--- Backups/vIRB4600-40-2.55-RW11/RAPID/TASK3/SYSMOD/RRC_Control_Rx.sys ---
MODULE RRC_Control_Rx(SYSMODULE)
    !***********************************************************************************
    !
    ! ETH Zurich / Robotic Fabrication Lab
    ! HIB C 13 / Stefano-Franscini-Platz 1
    ! CH-8093 Zurich
    !
    !***********************************************************************************
    !
    ! PROJECT     :  RRC - Rapid Robot Communication
    !
    ! FUNCTION    :  Control modul for the project
    !
    ! AUTHOR      :  Philippe Fleischmann
    !
    ! EMAIL       :  rrc@arch.ethz.ch
    !
    ! HISTORY     :  2019.02.22
    !
    ! Copyright   :  ETH Zurich (CH) 2019
    !                - Philippe Fleischmann
    !                - Michael Lyrenmann
    !                - Gonzalo Casas
    !
    ! License     :  This code base is governed by an EULA (End-User License Agreement)
    !                which you have received together with the software.
    !                You are not allowed to use the software on a real robots
    !                without a signed EULA.
    !
    !                A copy of the EULA content is in the controller task (T_CTRL).
    !
    !***********************************************************************************

    !************************************************
    ! Function    :     Main for Project RRC
    ! Programmer  :     Philippe Fleischmann
    ! Date        :     2019.02.22
    !***************** ETH Zurich *******************
    !
    PROC r_RRC_Main()
        !
        ! Wait until controller has set taskliste all
        WaitTime n_RRC_TimeTaskLiAll;
        !
        ! Task synchronisation
        WaitSyncTask id_RRC_MainSta,tl_RRC_All;
        !
        ! Message for Operator
        TPWrite "RRC Main";
        !
        ! Initialize cell
        r_RRC_InitCell;
        !
        ! Work process
        WHILE b_RRC_Run=TRUE DO
            !
            ! Check and receive data from client 1
            IF b_RRC_Com{n_RRC_R1_ChaNr}=TRUE r_RRC_CheckAndRecFrmClient n_RRC_R1_ChaNr;
            !
            ! Check and receive data from client 2
            IF b_RRC_Com{n_RRC_R2_ChaNr}=TRUE r_RRC_CheckAndRecFrmClient n_RRC_R2_ChaNr;
            !
            ! Check and receive data from client 3
            IF b_RRC_Com{n_RRC_R3_ChaNr}=TRUE r_RRC_CheckAndRecFrmClient n_RRC_R3_ChaNr;
            !
            ! Check and receive data from client 4
            IF b_RRC_Com{n_RRC_R4_ChaNr}=TRUE r_RRC_CheckAndRecFrmClient n_RRC_R4_ChaNr;
            !
            ! Check cycle time stop watch activ
            IF b_RRC_EvLogMsgInUntilMsgOutTime=TRUE THEN
                !
                ! Measure cycle time
                IF b_RRC_FeedbackOut=TRUE THEN
                    !
                    ! Reset variable
                    b_RRC_FeedbackOut:=FALSE;
                    !
                    ! Stop read message input to feedback done watch
                    ClkStop clk_RRC_MsgInUntilMsgOut;
                    !
                    ! Log current read and unpack time in RobotStudio output
                    r_RRC_EvLogMsg st_RRC_EvLogMsgHeader,"Msg in until Msg out time : "+NumToStr(ClkRead(clk_RRC_MsgInUntilMsgOut\HighRes),3);
                ENDIF
            ENDIF
        ENDWHILE
        !
        ! Message for Operator
        TPWrite "RRC End";
        !
        ! Task synchronisation
        WaitSyncTask id_RRC_MainEnd,tl_RRC_All;
        !
        RETURN ;
    ERROR
        ! Placeholder for Error Code...
    ENDPROC

    !************************************************
    ! Function    :     Initialize Cell
    ! Programmer  :     Philippe Fleischmann
    ! Date        :     2019.02.22
    !***************** ETH Zurich *******************
    !
    PROC r_RRC_InitCell()
        !
        ! Task synchronisation
        WaitSyncTask id_RRC_InitSta,tl_RRC_All;
        !
        ! Task synchronisation wait for controller data
        WaitSyncTask id_RRC_InitCtrl,tl_RRC_All;
        !
        ! Initialize variables
        r_RRC_InitVar;
        !
        ! Initalize protocol log
        !* r_RRC_LogProtInit;
        !
        ! Initialize sockets
        IF b_RRC_SocketActiv=TRUE r_RRC_InitSockets;
        !
        ! Task synchronisation
        WaitSyncTask id_RRC_InitEnd,tl_RRC_All;
        RETURN ;
    ERROR
        ! Placeholder for Error Code...
    ENDPROC

    !************************************************
    ! Function    :     Initialize Variables
    ! Programmer  :     Philippe Fleischmann
    ! Date        :     2019.02.22
    !***************** ETH Zurich *******************
    !
    PROC r_RRC_InitVar()
        !
        ! Set Task on
        b_RRC_TaskReceiverOn:=TRUE;
        !
        ! Reset buffer full bits controller
        b_RRC_BufFullMa{n_RRC_R1_ChaNr}:=FALSE;
        b_RRC_BufFullMa{n_RRC_R2_ChaNr}:=FALSE;
        b_RRC_BufFullMa{n_RRC_R3_ChaNr}:=FALSE;
        b_RRC_BufFullMa{n_RRC_R4_ChaNr}:=FALSE;
        !
        ! Reset buffer full bits robot
        b_RRC_BufFullRob{n_RRC_R1_ChaNr}:=FALSE;
        b_RRC_BufFullRob{n_RRC_R2_ChaNr}:=FALSE;
        b_RRC_BufFullRob{n_RRC_R3_ChaNr}:=FALSE;
        b_RRC_BufFullRob{n_RRC_R4_ChaNr}:=FALSE;
        !
        ! Set first cycle bools
        b_RRC_FirstProtocolAfterPPMain:=TRUE;
        !
        ! Temp to measure cycle time
        b_RRC_FeedbackOut:=FALSE;
        !
        ! Reset counters controller
        n_RRC_WritePtrBufCtrl{n_RRC_R1_ChaNr}:=0;
        n_RRC_WritePtrBufCtrl{n_RRC_R2_ChaNr}:=0;
        n_RRC_WritePtrBufCtrl{n_RRC_R3_ChaNr}:=0;
        n_RRC_WritePtrBufCtrl{n_RRC_R4_ChaNr}:=0;
        !
        ! Reset counters robot
        n_RRC_WritePtrBufRob{n_RRC_R1_ChaNr}:=0;
        n_RRC_WritePtrBufRob{n_RRC_R2_ChaNr}:=0;
        n_RRC_WritePtrBufRob{n_RRC_R3_ChaNr}:=0;
        n_RRC_WritePtrBufRob{n_RRC_R4_ChaNr}:=0;
        !
        ! Clear buffer controller
        FOR i FROM 1 TO DIM(bm_RRC_RecBufferCtrl,2) DO
            !
            ! Overwrite with an empty message
            bm_RRC_RecBufferCtrl{n_RRC_R1_ChaNr,i}:=bmEmpty;
            bm_RRC_RecBufferCtrl{n_RRC_R2_ChaNr,i}:=bmEmpty;
            bm_RRC_RecBufferCtrl{n_RRC_R3_ChaNr,i}:=bmEmpty;
            bm_RRC_RecBufferCtrl{n_RRC_R4_ChaNr,i}:=bmEmpty;
            !
        ENDFOR
        !
        ! Clear buffer robots
        FOR i FROM 1 TO DIM(bm_RRC_RecBufferRob,2) DO
            !
            ! Overwrite with an empty message
            bm_RRC_RecBufferRob{n_RRC_R1_ChaNr,i}:=bmEmpty;
            bm_RRC_RecBufferRob{n_RRC_R2_ChaNr,i}:=bmEmpty;
            bm_RRC_RecBufferRob{n_RRC_R3_ChaNr,i}:=bmEmpty;
            bm_RRC_RecBufferRob{n_RRC_R4_ChaNr,i}:=bmEmpty;
            !
        ENDFOR
        !
        ! Reset expected Sequince ID
        n_RRC_SIDExpected{n_RRC_R1_ChaNr}:=0;
        n_RRC_SIDExpected{n_RRC_R2_ChaNr}:=0;
        n_RRC_SIDExpected{n_RRC_R3_ChaNr}:=0;
        n_RRC_SIDExpected{n_RRC_R4_ChaNr}:=0;
        RETURN ;
    ERROR
        ! Placeholder for Error Code...
    ENDPROC

    !************************************************
    ! Function    :     ProgError
    ! Programmer  :     Philippe Fleischmann
    ! Date        :     2019.02.22
    !***************** ETH Zurich *******************
    !
    PROC r_RRC_ProgError()
        !
        ! User Info
        TPWrite "Program Error";
        !
        ! Stop Program
        Stop;
        RETURN ;
    ERROR
        ! Placeholder for Error Code...
    ENDPROC

ENDMODULE

--- Backups/vIRB4600-40-2.55-RW11/RAPID/TASK3/SYSMOD/RRC_DataTask_Rx.sys ---
MODULE RRC_DataTask_Rx(SYSMODULE)
    !***********************************************************************************
    !
    ! ETH Zurich / Robotic Fabrication Lab
    ! HIB C 13 / Stefano-Franscini-Platz 1
    ! CH-8093 Zurich
    !
    !***********************************************************************************
    !
    ! PROJECT     :  RRC - Rapid Robot Communication
    !
    ! FUNCTION    :  Includ all Task specific Data's
    !
    ! AUTHOR      :  Philippe Fleischmann
    !
    ! EMAIL       :  rrc@arch.ethz.ch
    !
    ! HISTORY     :  2019.02.22
    !
    ! Copyright   :  ETH Zurich (CH) 2019
    !                - Philippe Fleischmann
    !                - Michael Lyrenmann
    !                - Gonzalo Casas
    !
    ! License     :  This code base is governed by an EULA (End-User License Agreement)
    !                which you have received together with the software.
    !                You are not allowed to use the software on a real robots
    !                without a signed EULA.
    !
    !                A copy of the EULA content is in the controller task (T_CTRL).
    !
    !***********************************************************************************

    !************************************************
    ! Declaration :     bool
    !************************************************
    !
    CONST bool b_RRC_Run:=TRUE;
    !
    TASK PERS bool b_RRC_SocketActiv:=TRUE;
    TASK PERS bool b_RRC_PrintPrio1:=FALSE;
    TASK PERS bool b_RRC_PrintPrio2:=FALSE;
    !
    TASK PERS bool b_RRC_BufFullMa{n_RRC_NumOfCha}:=[FALSE,FALSE,FALSE,FALSE];
    TASK PERS bool b_RRC_BufFullRob{n_RRC_NumOfCha}:=[FALSE,FALSE,FALSE,FALSE];
    TASK PERS bool b_RRC_LogHelper{n_RRC_NumOfCha}:=[FALSE,FALSE,FALSE,FALSE];
    !
    TASK PERS bool b_RRC_FirstProtocolAfterPPMain:=FALSE;

    !************************************************
    ! Declaration :     num
    !************************************************
    !
    CONST num n_RRC_NumOfCha:=4;
    CONST num n_RRC_RecMinData:=49;
    CONST num n_RRC_NoOfByMsgLen:=4;
    CONST num n_RRC_TimeOutRecRobSocRec:=10;
    !
    TASK PERS num n_RRC_WritePtrBufCtrl{n_RRC_NumOfCha}:=[0,0,0,0];
    TASK PERS num n_RRC_WritePtrBufRob{n_RRC_NumOfCha}:=[7,0,0,0];
    TASK PERS num n_RRC_SIDExpected{n_RRC_NumOfCha}:=[1,0,0,0];
    TASK PERS num n_RRC_SIDIs{n_RRC_NumOfCha}:=[70001,0,0,0];
    !
    VAR num n_RRC_MsgLenRob{n_RRC_NumOfCha};
    VAR num n_RRC_NoOfRecBytesRob{n_RRC_NumOfCha};

    !************************************************
    ! Declaration :     string
    !************************************************
    !
    TASK PERS string st_RRC_EvLogMsgHeader:="RRC -- Receiver";
    TASK PERS string st_RRC_SIDRestart:="S-ID User code restarted";
    !
    TASK PERS string st_RRC_UIAnswer:="Stop";
    TASK PERS string st_RRC_ActMsg1:="Expected protocol version: 1.0";
    TASK PERS string st_RRC_ActMsg2:="Received protocol version: 2.0";
    TASK PERS string st_RRC_ActMsg3:="Expected: 2";
    TASK PERS string st_RRC_ActMsg4:="Received: 70001";
    TASK PERS string st_RRC_ActMsg5:="";
    TASK PERS string st_RRC_ActBtn1:="Stop";
    TASK PERS string st_RRC_ActBtn2:="100 mm/s";
    TASK PERS string st_RRC_ActBtn3:="Set my Speed";
    TASK PERS string st_RRC_ActBtn4:="";
    TASK PERS string st_RRC_ActBtn5:="";
    TASK PERS string st_RRC_Header:="Protocol mismatch";
    !
    VAR string st_RRC_IP_ClientRec{n_RRC_NumOfCha}:=["","","",""];

    !************************************************
    ! Declaration :     clock
    !************************************************
    !
    VAR clock clk_RRC_ReadAndUnpack;
    VAR clock clk_RRC_MsgInUntilMsgOut;

    !************************************************
    ! Declaration :     RRC_Protokol
    !************************************************
    !
    CONST RRC_Protocol pro_RRC_Empty:=[[0,0,0,0],[0,0,0,"",0,0,"",0,0,0,"",0,"",0,"",0,"",0,"",0,"",0,"",0,"",0,0,0,0,0,0,0,0,0,0,0,0,0,0,0,0,0,0,0,0,0,0,0,0,0,0,0,0,0,0,0,0,0,0,0,0,0]];
    !
    VAR RRC_Protocol pro_RRC_ActMsgRob:=[[0,0,0,0],[0,0,0,"",0,0,"",0,0,0,"",0,"",0,"",0,"",0,"",0,"",0,"",0,"",0,0,0,0,0,0,0,0,0,0,0,0,0,0,0,0,0,0,0,0,0,0,0,0,0,0,0,0,0,0,0,0,0,0,0,0,0]];
    !
    TASK PERS RRC_Protocol pro_RRC_ActMsgTemp:=[[0,0,0,0],[0,0,0,"",0,0,"",0,0,0,"",0,"",0,"",0,"",0,"",0,"",0,"",0,"",0,0,0,0,0,0,0,0,0,0,0,0,0,0,0,0,0,0,0,0,0,0,0,0,0,0,0,0,0,0,0,0,0,0,0,0,0]];
    !
    TASK PERS RRC_Protocol pro_RRC_ActMsgRec{n_RRC_NumOfCha}:=[
    [[63,2,1.67742E+9,464],[1,0,15,"r_RRC_GetJoints",1,0,"",0,0,0,"",0,"",0,"",0,"",0,"",0,"",0,"",0,"",0,0,0,0,0,0,0,0,0,0,0,0,0,0,0,0,0,0,0,0,0,0,0,0,0,0,0,0,0,0,0,0,0,0,0,0,0]],
    [[67,4,1.58281E+9,242],[4,0,15,"r_RRC_WaitTime",1,0,"",0,0,24,"E-Level Channel 2 Controller",0,"",0,"",0,"",0,"",0,"",0,"",0,"",1,1,0,0,0,0,0,0,0,0,0,0,0,0,0,0,0,0,0,0,0,0,0,0,0,0,0,0,0,0,0,0,0,0,0,0,0]],
    [[120,4,1.55775E+9,695],[11,0,12,"r_RRC_MoveL",1,0,"",0,0,0,"",0,"",0,"",0,"",0,"",0,"",0,"",0,"",15,542.04,-200,237.57,0,0,1,0,28000,-3400,-3138,0,0,0,230,20,0,0,0,0,0,0,0,0,0,0,0,0,0,0,0,0,0,0,0,0,0]],
    [[120,4,1.55775E+9,695],[11,0,12,"r_RRC_MoveL",1,0,"",0,0,0,"",0,"",0,"",0,"",0,"",0,"",0,"",0,"",15,542.04,-200,237.57,0,0,1,0,28000,-3400,-3138,0,0,0,230,20,0,0,0,0,0,0,0,0,0,0,0,0,0,0,0,0,0,0,0,0,0]]];

    !************************************************
    ! Declaration :     rawbytes
    !************************************************
    !
    VAR rawbytes rb_RRC_BufferMsgLenRob{n_RRC_NumOfCha};
    VAR rawbytes rb_RRC_BufferRob{n_RRC_NumOfCha};

    !************************************************
    ! Declaration :     socketdev
    !************************************************
    !
    VAR socketdev sod_RRC_ServerRec{n_RRC_NumOfCha};
    VAR socketdev sod_RRC_ClientRec{n_RRC_NumOfCha};

    !************************************************
    ! Declaration :     RRC_buffer_msg
    !************************************************
    !
    CONST RRC_buffer_msg bmEmpty:=[[0,0,0,"",0,0,"",0,0,0,"",0,"",0,"",0,"",0,"",0,"",0,"",0,"",0,0,0,0,0,0,0,0,0,0,0,0,0,0,0,0,0,0,0,0,0,0,0,0,0,0,0,0,0,0,0,0,0,0,0,0,0],FALSE];
ENDMODULE

--- Backups/vIRB4600-40-2.55-RW11/RAPID/TASK3/SYSMOD/RRC_Log_Rx.sys ---
MODULE RRC_Log_Rx(SYSMODULE)
    !***********************************************************************************
    !
    ! ETH Zurich / Robotic Fabrication Lab
    ! HIB C 13 / Stefano-Franscini-Platz 1
    ! CH-8093 Zurich
    !
    !***********************************************************************************
    !
    ! PROJECT     :  RRC - Rapid Robot Communication
    !
    ! FUNCTION    :  Inclouds all logger functions
    !
    ! AUTHOR      :  Philippe Fleischmann
    !
    ! EMAIL       :  rrc@arch.ethz.ch
    !
    ! HISTORY     :  2019.02.22
    !
    ! Copyright   :  ETH Zurich (CH) 2019
    !                - Philippe Fleischmann
    !                - Michael Lyrenmann
    !                - Gonzalo Casas
    !
    ! License     :  This code base is governed by an EULA (End-User License Agreement)
    !                which you have received together with the software.
    !                You are not allowed to use the software on a real robots
    !                without a signed EULA.
    !
    !                A copy of the EULA content is in the controller task (T_CTRL).
    !
    !***********************************************************************************

    !************************************************
    ! Declaration :     bool
    !************************************************
    !
    CONST bool b_RRC_LogActiv:=TRUE;

    !************************************************
    ! Declaration :     num
    !************************************************
    !
    TASK PERS num n_RRC_LogMsgCountr:=0;
    TASK PERS num n_RRC_FileNr:=1;
    CONST num n_RRC_LogMaxMsg:=1000000;

    !************************************************
    ! Declaration :     string
    !************************************************
    !
    CONST string st_RRC_LogDirPathRC:="RemovableDisk1:RRC_Log/";
    CONST string st_RRC_LogDirPathVC:="Home:/RRC_Log/";
    TASK PERS string st_RRC_LogDirPath:="RemovableDisk1:RRC_Log/";
    CONST string st_RRC_LogFileName:="RRC_LogReceiver";
    CONST string st_RRC_LogFileFormat:=".csv";
    CONST string st_RRC_LogProgrammer:="Philipppe Fleischmann";
    !
    CONST string stTab:="\09";

    ! Global System Data
    TASK PERS string st_RFL_SystemDate:="2018-06-28";
    TASK PERS string st_RFL_SystemTime:="15:49:26";

    !************************************************
    ! Declaration :     iodev
    !************************************************
    !
    VAR iodev iodev_RRC_LogFile;

    !************************************************
    ! Declaration :     dir
    !************************************************
    !
    VAR dir dir_RRC_Dev;

    !************************************************
    ! Declaration :     clock
    !************************************************
    !
    VAR clock ck_RRC_LogTimer;

    !************************************************
    ! Discription :     Steps for log integration in code
    ! Programmer  :     Philippe Fleischmann
    ! Date        :     2019.02.22
    !***************** ETH Zurich *******************
    !
    ! 1. Create a log folder, run the procedure manuali PP to Routine
    !* r_RRC_CrateLogFolder;
    !
    ! 2. Integrate Initialzie log function
    !* r_RRC_LogInit
    !
    ! 3. Integrate write log
    !* IF b_RRC_LogActiv=TRUE r_RRC_LogWriteRhinoMsg message_command;
    !
    ! 4. Integrate Close file (when posible)
    !* IF b_RRC_LogActiv=TRUE r_RRC_LogFileClose;
    !
    !************************************************

    !************************************************
    ! Function    :     Log initialization
    ! Programmer  :     Philippe Fleischmann
    ! Date        :     2019.02.22
    !***************** ETH Zurich *******************
    !
    PROC r_RRC_LogTest()
        !
        ! Initialize logfile
        r_RRC_LogProtInit;
        !
        ! Load protocol message
        ! Header
        pro_RRC_ActMsgRob.ProtocolHeader.M_Len:=104;
        pro_RRC_ActMsgRob.ProtocolHeader.Ver:=1;
        pro_RRC_ActMsgRob.ProtocolHeader.TS_Sec:=33;
        pro_RRC_ActMsgRob.ProtocolHeader.TS_NSec:=399;
        !
        ! Main data
        pro_RRC_ActMsgRob.ProtocolData.S_ID:=300;
        pro_RRC_ActMsgRob.ProtocolData.E_Lev:=0;
        pro_RRC_ActMsgRob.ProtocolData.F_Lev:=1;
        pro_RRC_ActMsgRob.ProtocolData.I_Len:=8;
        pro_RRC_ActMsgRob.ProtocolData.Instr:="MoveAbsJ";
        pro_RRC_ActMsgRob.ProtocolData.F_Len:=4;
        pro_RRC_ActMsgRob.ProtocolData.Feedb:="Done";
        pro_RRC_ActMsgRob.ProtocolData.F_ID:=300;
        !
        ! String parameter
        pro_RRC_ActMsgRob.ProtocolData.St_Cnt:=5;
        pro_RRC_ActMsgRob.ProtocolData.St1_Len:=4;
        pro_RRC_ActMsgRob.ProtocolData.St1:="This";
        pro_RRC_ActMsgRob.ProtocolData.St2_Len:=2;
        pro_RRC_ActMsgRob.ProtocolData.St2:="is";
        pro_RRC_ActMsgRob.ProtocolData.St3_Len:=1;
        pro_RRC_ActMsgRob.ProtocolData.St3:="a";
        pro_RRC_ActMsgRob.ProtocolData.St4_Len:=8;
        pro_RRC_ActMsgRob.ProtocolData.St4:="protocol";
        pro_RRC_ActMsgRob.ProtocolData.St5_Len:=5;
        pro_RRC_ActMsgRob.ProtocolData.St5:="test";
        !
        ! Value parameter
        pro_RRC_ActMsgRob.ProtocolData.V_Cnt:=1;
        pro_RRC_ActMsgRob.ProtocolData.V1:=99;
        FOR i FROM 1 TO 1 DO


            r_RRC_LogPro pro_RRC_ActMsgRob;

        ENDFOR

        Close iodev_RRC_LogFile;

        Stop;

        RETURN ;
    ERROR
    ENDPROC

    !************************************************
    ! Function    :     Initialize protocol log
    ! Programmer  :     Philippe Fleischmann
    ! Date        :     2019.02.22
    !***************** ETH Zurich *******************
    !
    PROC r_RRC_LogProtInit()
        !
        ! Selcet the writ path for the log file
        IF RobOS()=TRUE THEN
            !
            ! Real controller write to MemoryStick
            st_RRC_LogDirPath:=st_RRC_LogDirPathRC;
        ELSE
            !
            ! Virtual controller write to Home
            st_RRC_LogDirPath:=st_RRC_LogDirPathVC;
        ENDIF
        !
        ! Initalize variables
        n_RRC_LogMsgCountr:=0;
        !
        ! Opent directory
        OpenDir dir_RRC_Dev,st_RRC_LogDirPath;
        !
        ! Check for log file
        IF IsFile(st_RRC_LogDirPath+st_RRC_LogFileName+st_RRC_LogFileFormat) THEN
            !
            ! Remove the old log file
            RemoveFile st_RRC_LogDirPath+st_RRC_LogFileName+st_RRC_LogFileFormat;
        ENDIF
        !
        ! Create and open a new log file
        Open st_RRC_LogDirPath+st_RRC_LogFileName+st_RRC_LogFileFormat,iodev_RRC_LogFile\Write;
        !
        ! Write column title for
        Write iodev_RRC_LogFile,"L-Nr;LogTime;LogFormat;"\NoNewLine;
        Write iodev_RRC_LogFile,"M_Len;Ver;TS-Sec;TS-NSec;"\NoNewLine;
        Write iodev_RRC_LogFile,"S_ID;E_Lev;I_Len;Instr;F_Lev;F_Len;Feedb;F_ID;"\NoNewLine;
        Write iodev_RRC_LogFile,"St_Ctr;St1_Len;St1;St2_Len;St2;St3_Len;St3;St4_Len;St4;St5_Len;St5;"\NoNewLine;
        Write iodev_RRC_LogFile,"V_Ctr;V1;V2;V3;V4;V5;V6;V7;V8;V9;V10;"\NoNewLine;
        Write iodev_RRC_LogFile,"V11;V12;V13;V14;V15;V16;V17;V18;V19;V20;"\NoNewLine;
        Write iodev_RRC_LogFile,"V21;V22;V23;V24;V25;V26;V27;V28;V29;V30;";
        !
        ! Reset and start log timer
        ClkReset ck_RRC_LogTimer;
        ClkStart ck_RRC_LogTimer;
        !
        ! Log message
        r_RRC_EvLogMsg st_RRC_LogFileName,"Log inititalizaion, done";
        RETURN ;
    ERROR
        !
        ! Handle error open directory
        IF ERRNO=ERR_FILEACC THEN
            !
            ! Create the log folder
            MakeDir st_RRC_LogDirPath;
            !
            ! Log message
            r_RRC_EvLogMsg st_RRC_LogFileName,"Log Directory created";
            !
            ! Retyry to open directory
            RETRY;
        ENDIF
        Stop;
        Stop;
    ENDPROC

    !************************************************
    ! Function    :     Log protocol
    ! Programmer  :     Philippe Fleischmann
    ! Date        :     2019.02.22
    !***************** ETH Zurich *******************
    !
    PROC r_RRC_LogPro(RRC_Protocol proMsg)
        !
        ! Increuse log message counter
        Incr n_RRC_LogMsgCountr;
        !
        ! Log only until max message is reached
        IF n_RRC_LogMsgCountr<=n_RRC_LogMaxMsg THEN
            !
            ! Add counter nuber and time
            Write iodev_RRC_LogFile,NumToStr(n_RRC_LogMsgCountr,0)+";"\NoNewLine;
            Write iodev_RRC_LogFile,NumToStr(ClkRead(ck_RRC_LogTimer\HighRes),3)+";"\NoNewLine;
            !
            ! Add log format
            Write iodev_RRC_LogFile,"protocol"+";"\NoNewLine;
            !
            ! Add protocol header
            Write iodev_RRC_LogFile,NumToStr(proMsg.ProtocolHeader.M_Len,0)+";"\NoNewLine;
            Write iodev_RRC_LogFile,NumToStr(proMsg.ProtocolHeader.Ver,0)+";"\NoNewLine;
            Write iodev_RRC_LogFile,NumToStr(proMsg.ProtocolHeader.TS_Sec,0)+";"\NoNewLine;
            Write iodev_RRC_LogFile,NumToStr(proMsg.ProtocolHeader.TS_NSec,3)+";"\NoNewLine;
            !
            ! Protocol main data
            Write iodev_RRC_LogFile,NumToStr(proMsg.ProtocolData.S_ID,0)+";"\NoNewLine;
            Write iodev_RRC_LogFile,NumToStr(proMsg.ProtocolData.E_Lev,0)+";"\NoNewLine;
            Write iodev_RRC_LogFile,NumToStr(proMsg.ProtocolData.I_Len,0)+";"\NoNewLine;
            Write iodev_RRC_LogFile,proMsg.ProtocolData.Instr+";"\NoNewLine;
            Write iodev_RRC_LogFile,NumToStr(proMsg.ProtocolData.F_Lev,0)+";"\NoNewLine;
            Write iodev_RRC_LogFile,NumToStr(proMsg.ProtocolData.F_Len,0)+";"\NoNewLine;
            Write iodev_RRC_LogFile,proMsg.ProtocolData.Feedb+";"\NoNewLine;
            Write iodev_RRC_LogFile,NumToStr(proMsg.ProtocolData.F_ID,0)+";"\NoNewLine;
            !
            ! Protocol string parameter
            Write iodev_RRC_LogFile,NumToStr(proMsg.ProtocolData.St_Cnt,0)+";"\NoNewLine;
            Write iodev_RRC_LogFile,NumToStr(proMsg.ProtocolData.St1_Len,0)+";"\NoNewLine;
            Write iodev_RRC_LogFile,proMsg.ProtocolData.St1+";"\NoNewLine;
            Write iodev_RRC_LogFile,NumToStr(proMsg.ProtocolData.St2_Len,0)+";"\NoNewLine;
            Write iodev_RRC_LogFile,proMsg.ProtocolData.St2+";"\NoNewLine;
            Write iodev_RRC_LogFile,NumToStr(proMsg.ProtocolData.St3_Len,0)+";"\NoNewLine;
            Write iodev_RRC_LogFile,proMsg.ProtocolData.St3+";"\NoNewLine;
            Write iodev_RRC_LogFile,NumToStr(proMsg.ProtocolData.St4_Len,0)+";"\NoNewLine;
            Write iodev_RRC_LogFile,proMsg.ProtocolData.St4+";"\NoNewLine;
            Write iodev_RRC_LogFile,NumToStr(proMsg.ProtocolData.St5_Len,0)+";"\NoNewLine;
            Write iodev_RRC_LogFile,proMsg.ProtocolData.St5+";"\NoNewLine;
            !
            ! Protocol value parameter
            Write iodev_RRC_LogFile,NumToStr(proMsg.ProtocolData.V_Cnt,0)+";"\NoNewLine;
            Write iodev_RRC_LogFile,NumToStr(proMsg.ProtocolData.V1,3)+";"\NoNewLine;
            Write iodev_RRC_LogFile,NumToStr(proMsg.ProtocolData.V2,3)+";"\NoNewLine;
            Write iodev_RRC_LogFile,NumToStr(proMsg.ProtocolData.V3,3)+";"\NoNewLine;
            Write iodev_RRC_LogFile,NumToStr(proMsg.ProtocolData.V4,3)+";"\NoNewLine;
            Write iodev_RRC_LogFile,NumToStr(proMsg.ProtocolData.V5,3)+";"\NoNewLine;
            Write iodev_RRC_LogFile,NumToStr(proMsg.ProtocolData.V6,3)+";"\NoNewLine;
            Write iodev_RRC_LogFile,NumToStr(proMsg.ProtocolData.V7,3)+";"\NoNewLine;
            Write iodev_RRC_LogFile,NumToStr(proMsg.ProtocolData.V8,3)+";"\NoNewLine;
            Write iodev_RRC_LogFile,NumToStr(proMsg.ProtocolData.V9,3)+";"\NoNewLine;
            Write iodev_RRC_LogFile,NumToStr(proMsg.ProtocolData.V10,3)+";"\NoNewLine;
            Write iodev_RRC_LogFile,NumToStr(proMsg.ProtocolData.V11,3)+";"\NoNewLine;
            Write iodev_RRC_LogFile,NumToStr(proMsg.ProtocolData.V12,3)+";"\NoNewLine;
            Write iodev_RRC_LogFile,NumToStr(proMsg.ProtocolData.V13,3)+";"\NoNewLine;
            Write iodev_RRC_LogFile,NumToStr(proMsg.ProtocolData.V14,3)+";"\NoNewLine;
            Write iodev_RRC_LogFile,NumToStr(proMsg.ProtocolData.V15,3)+";"\NoNewLine;
            Write iodev_RRC_LogFile,NumToStr(proMsg.ProtocolData.V16,3)+";"\NoNewLine;
            Write iodev_RRC_LogFile,NumToStr(proMsg.ProtocolData.V17,3)+";"\NoNewLine;
            Write iodev_RRC_LogFile,NumToStr(proMsg.ProtocolData.V18,3)+";"\NoNewLine;
            Write iodev_RRC_LogFile,NumToStr(proMsg.ProtocolData.V19,3)+";"\NoNewLine;
            Write iodev_RRC_LogFile,NumToStr(proMsg.ProtocolData.V20,3)+";"\NoNewLine;
            Write iodev_RRC_LogFile,NumToStr(proMsg.ProtocolData.V21,3)+";"\NoNewLine;
            Write iodev_RRC_LogFile,NumToStr(proMsg.ProtocolData.V22,3)+";"\NoNewLine;
            Write iodev_RRC_LogFile,NumToStr(proMsg.ProtocolData.V23,3)+";"\NoNewLine;
            Write iodev_RRC_LogFile,NumToStr(proMsg.ProtocolData.V24,3)+";"\NoNewLine;
            Write iodev_RRC_LogFile,NumToStr(proMsg.ProtocolData.V25,3)+";"\NoNewLine;
            Write iodev_RRC_LogFile,NumToStr(proMsg.ProtocolData.V26,3)+";"\NoNewLine;
            Write iodev_RRC_LogFile,NumToStr(proMsg.ProtocolData.V27,3)+";"\NoNewLine;
            Write iodev_RRC_LogFile,NumToStr(proMsg.ProtocolData.V28,3)+";"\NoNewLine;
            Write iodev_RRC_LogFile,NumToStr(proMsg.ProtocolData.V29,3)+";"\NoNewLine;
            Write iodev_RRC_LogFile,NumToStr(proMsg.ProtocolData.V30,3)+";"\NoNewLine;
            !
            ! Protocol end
            Write iodev_RRC_LogFile,";";
        ENDIF


        RETURN ;
    ERROR
        ! Placeholder for Error Code...
    ENDPROC

ENDMODULE

--- Backups/vIRB4600-40-2.55-RW11/RAPID/TASK4/SYSMOD/RRC_Control_Tx.sys ---
MODULE RRC_Control_Tx(SYSMODULE)
    !***********************************************************************************
    !
    ! ETH Zurich / Robotic Fabrication Lab
    ! HIB C 13 / Stefano-Franscini-Platz 1
    ! CH-8093 Zurich
    !
    !***********************************************************************************
    !
    ! PROJECT     :  RRC - Rapid Robot Communication
    !
    ! FUNCTION    :  Control modul for the project
    !
    ! AUTHOR      :  Philippe Fleischmann
    !
    ! EMAIL       :  rrc@arch.ethz.ch
    !
    ! HISTORY     :  2019.02.22
    !
    ! Copyright   :  ETH Zurich (CH) 2019
    !                - Philippe Fleischmann
    !                - Michael Lyrenmann
    !                - Gonzalo Casas
    !
    ! License     :  This code base is governed by an EULA (End-User License Agreement)
    !                which you have received together with the software.
    !                You are not allowed to use the software on a real robots
    !                without a signed EULA.
    !
    !                A copy of the EULA content is in the controller task (T_CTRL).
    !
    !***********************************************************************************

    !************************************************
    ! Function    :     Main for Project RRC
    ! Programmer  :     Philippe Fleischmann
    ! Date        :     2019.02.22
    !***************** ETH Zurich *******************
    !
    PROC r_RRC_Main()
        !
        ! Wait until controller has set taskliste all
        WaitTime n_RRC_TimeTaskLiAll;
        !
        ! Task synchronisation
        WaitSyncTask id_RRC_MainSta,tl_RRC_All;
        !
        ! Message for Operator
        TPWrite "RRC Main";
        !
        ! Inititalize cell
        r_RRC_InitCell;
        !
        ! Work process
        WHILE b_RRC_Run=TRUE DO
            !
            ! Check and send data to client
            IF b_RRC_Com{n_RRC_R1_ChaNr}=TRUE THEN
                !
                ! For robot
                IF bm_RRC_SenBufferRob{n_RRC_R1_ChaNr,n_RRC_ReadPtrSenBufRob{n_RRC_R1_ChaNr}}.startbit=TRUE r_RRC_PackSendDataToClient\Rob,n_RRC_R1_ChaNr;
                !
                ! For controller
                IF bm_RRC_SenBufferCtrl{n_RRC_R1_ChaNr,n_RRC_ReadPtrSenBufCtrl{n_RRC_R1_ChaNr}}.startbit=TRUE r_RRC_PackSendDataToClient\Ctrl,n_RRC_R1_ChaNr;
            ENDIF
            !
            ! Check and send data to client
            IF b_RRC_Com{n_RRC_R2_ChaNr}=TRUE THEN
                !
                ! For robot
                IF bm_RRC_SenBufferRob{n_RRC_R2_ChaNr,n_RRC_ReadPtrSenBufRob{n_RRC_R2_ChaNr}}.startbit=TRUE r_RRC_PackSendDataToClient\Rob,n_RRC_R2_ChaNr;
                !
                ! For controller
                IF bm_RRC_SenBufferCtrl{n_RRC_R2_ChaNr,n_RRC_ReadPtrSenBufCtrl{n_RRC_R2_ChaNr}}.startbit=TRUE r_RRC_PackSendDataToClient\Ctrl,n_RRC_R2_ChaNr;
            ENDIF
            !
            ! Check and send data to client
            IF b_RRC_Com{n_RRC_R3_ChaNr}=TRUE THEN
                !
                ! For robot
                IF bm_RRC_SenBufferRob{n_RRC_R3_ChaNr,n_RRC_ReadPtrSenBufRob{n_RRC_R3_ChaNr}}.startbit=TRUE r_RRC_PackSendDataToClient\Rob,n_RRC_R3_ChaNr;
                !
                ! For controller
                IF bm_RRC_SenBufferCtrl{n_RRC_R3_ChaNr,n_RRC_ReadPtrSenBufCtrl{n_RRC_R3_ChaNr}}.startbit=TRUE r_RRC_PackSendDataToClient\Ctrl,n_RRC_R3_ChaNr;
            ENDIF
            !
            ! Check and send data to client
            IF b_RRC_Com{n_RRC_R4_ChaNr}=TRUE THEN
                !
                ! For robot
                IF bm_RRC_SenBufferRob{n_RRC_R4_ChaNr,n_RRC_ReadPtrSenBufRob{n_RRC_R4_ChaNr}}.startbit=TRUE r_RRC_PackSendDataToClient\Rob,n_RRC_R4_ChaNr;
                !
                ! For controller
                IF bm_RRC_SenBufferCtrl{n_RRC_R4_ChaNr,n_RRC_ReadPtrSenBufCtrl{n_RRC_R4_ChaNr}}.startbit=TRUE r_RRC_PackSendDataToClient\Ctrl,n_RRC_R4_ChaNr;
            ENDIF
        ENDWHILE
        !
        ! Message for Operator
        TPWrite "RRC End";
        !
        ! Task synchronisation
        WaitSyncTask id_RRC_MainEnd,tl_RRC_All;
        !
        RETURN ;
    ERROR
        ! Placeholder for Error Code...
    ENDPROC

    !************************************************
    ! Function    :     Initialize Cell
    ! Programmer  :     Philippe Fleischmann
    ! Date        :     2019.02.22
    !***************** ETH Zurich *******************
    !
    PROC r_RRC_InitCell()
        !
        ! Task synchronisation
        WaitSyncTask id_RRC_InitSta,tl_RRC_All;
        !
        ! Task synchronisation wait for controller data
        WaitSyncTask id_RRC_InitCtrl,tl_RRC_All;
        !
        ! Initialize variables
        r_RRC_InitVar;
        !
        ! Initialize sockets
        IF b_RRC_SocketActiv=TRUE r_RRC_InitSockets;
        !
        ! Task synchronisation
        WaitSyncTask id_RRC_InitEnd,tl_RRC_All;
        RETURN ;
    ERROR
        ! Placeholder for Error Code...
    ENDPROC

    !************************************************
    ! Function    :     Initialize Variables
    ! Programmer  :     Philippe Fleischmann
    ! Date        :     2019.02.22
    !***************** ETH Zurich *******************
    !
    PROC r_RRC_InitVar()
        !
        ! Set Task on
        b_RRC_TaskSenderOn:=TRUE;
        !
        ! Reset and start timestamp
        ClkReset clk_RRC_TimeStamp;
        ClkStart clk_RRC_TimeStamp;
        !
        ! Reset Counters
        n_RRC_WritePtrSenBufCtrl{n_RRC_R1_ChaNr}:=0;
        n_RRC_WritePtrSenBufCtrl{n_RRC_R2_ChaNr}:=0;
        n_RRC_WritePtrSenBufCtrl{n_RRC_R3_ChaNr}:=0;
        n_RRC_WritePtrSenBufCtrl{n_RRC_R4_ChaNr}:=0;
        !
        n_RRC_WritePtrSenBufRob{n_RRC_R1_ChaNr}:=0;
        n_RRC_WritePtrSenBufRob{n_RRC_R2_ChaNr}:=0;
        n_RRC_WritePtrSenBufRob{n_RRC_R3_ChaNr}:=0;
        n_RRC_WritePtrSenBufRob{n_RRC_R4_ChaNr}:=0;
        !
        n_RRC_ReadPtrSenBufCtrl{n_RRC_R1_ChaNr}:=1;
        n_RRC_ReadPtrSenBufCtrl{n_RRC_R2_ChaNr}:=1;
        n_RRC_ReadPtrSenBufCtrl{n_RRC_R3_ChaNr}:=1;
        n_RRC_ReadPtrSenBufCtrl{n_RRC_R4_ChaNr}:=1;
        !
        n_RRC_ReadPtrSenBufRob{n_RRC_R1_ChaNr}:=1;
        n_RRC_ReadPtrSenBufRob{n_RRC_R2_ChaNr}:=1;
        n_RRC_ReadPtrSenBufRob{n_RRC_R3_ChaNr}:=1;
        n_RRC_ReadPtrSenBufRob{n_RRC_R4_ChaNr}:=1;
        !
        n_RRC_SenHeaderSqzNr{n_RRC_R1_ChaNr}:=0;
        n_RRC_SenHeaderSqzNr{n_RRC_R2_ChaNr}:=0;
        n_RRC_SenHeaderSqzNr{n_RRC_R3_ChaNr}:=0;
        n_RRC_SenHeaderSqzNr{n_RRC_R4_ChaNr}:=0;
        !
        ! Clear Buffers
        FOR i FROM 1 TO DIM(bm_RRC_SenBufferCtrl,2) DO
            !
            ! Overwrite with an empty message
            bm_RRC_SenBufferCtrl{n_RRC_R1_ChaNr,i}:=bmEmpty;
            bm_RRC_SenBufferCtrl{n_RRC_R2_ChaNr,i}:=bmEmpty;
            bm_RRC_SenBufferCtrl{n_RRC_R3_ChaNr,i}:=bmEmpty;
            bm_RRC_SenBufferCtrl{n_RRC_R4_ChaNr,i}:=bmEmpty;
        ENDFOR
        !
        ! Clear Buffers
        FOR i FROM 1 TO DIM(bm_RRC_SenBufferRob,2) DO
            !
            ! Overwrite with an empty message
            bm_RRC_SenBufferRob{n_RRC_R1_ChaNr,i}:=bmEmpty;
            bm_RRC_SenBufferRob{n_RRC_R2_ChaNr,i}:=bmEmpty;
            bm_RRC_SenBufferRob{n_RRC_R3_ChaNr,i}:=bmEmpty;
            bm_RRC_SenBufferRob{n_RRC_R4_ChaNr,i}:=bmEmpty;
        ENDFOR
        !
        ! Clear Buffers
        FOR i FROM 1 TO DIM(pro_RRC_ActMsgSen,2) DO
            !
            ! Overwrite with an empty protocol
            pro_RRC_ActMsgSen{1,i}:=proEmpty;
            pro_RRC_ActMsgSen{1,i}:=proEmpty;
            pro_RRC_ActMsgSen{1,i}:=proEmpty;
            pro_RRC_ActMsgSen{1,i}:=proEmpty;
            !
            pro_RRC_ActMsgSen{2,i}:=proEmpty;
            pro_RRC_ActMsgSen{2,i}:=proEmpty;
            pro_RRC_ActMsgSen{2,i}:=proEmpty;
            pro_RRC_ActMsgSen{2,i}:=proEmpty;
        ENDFOR
        RETURN ;
    ERROR
        ! Placeholder for Error Code...
    ENDPROC

    !************************************************
    ! Function    :     ProgError
    ! Programmer  :     Philippe Fleischmann
    ! Date        :     2019.02.22
    !***************** ETH Zurich *******************
    !
    PROC r_RRC_ProgError()
        !
        ! User Info
        TPWrite "Program Error";
        !
        ! Stop Program
        Stop;
        RETURN ;
    ERROR
        ! Placeholder for Error Code...
    ENDPROC

ENDMODULE

--- Backups/vIRB4600-40-2.55-RW11/RAPID/TASK4/SYSMOD/RRC_DataTask_Tx.sys ---
MODULE RRC_DataTask_Tx(SYSMODULE)
    !***********************************************************************************
    !
    ! ETH Zurich / Robotic Fabrication Lab
    ! HIB C 13 / Stefano-Franscini-Platz 1
    ! CH-8093 Zurich
    !
    !***********************************************************************************
    !
    ! PROJECT     :  RRC - Rapid Robot Communication
    !
    ! FUNCTION    :  Includ all Task specific Data's
    !
    ! AUTHOR      :  Philippe Fleischmann
    !
    ! EMAIL       :  rrc@arch.ethz.ch
    !
    ! HISTORY     :  2019.02.22
    !
    ! Copyright   :  ETH Zurich (CH) 2019
    !                - Philippe Fleischmann
    !                - Michael Lyrenmann
    !                - Gonzalo Casas
    !
    ! License     :  This code base is governed by an EULA (End-User License Agreement)
    !                which you have received together with the software.
    !                You are not allowed to use the software on a real robots
    !                without a signed EULA.
    !
    !                A copy of the EULA content is in the controller task (T_CTRL).
    !
    !***********************************************************************************

    !************************************************
    ! Declaration :     bool
    !************************************************
    !
    CONST bool b_RRC_Run:=TRUE;
    !
    TASK PERS bool b_RRC_PrintPrio1:=FALSE;
    !
    TASK PERS bool b_RRC_SocketActiv:=TRUE;

    !************************************************
    ! Declaration :     num
    !************************************************
    !
    CONST num n_RRC_NumOfCha:=4;
    CONST num n_RRC_SenMinData:=1;
    CONST num n_RRC_NoOfByMsgLen:=4;
    CONST num n_RRC_SenHeaderMaxSqzNrRob:=1000000;
    CONST num n_RRC_ProtocolCtrl:=1;
    CONST num n_RRC_ProtocolRob:=2;
    CONST num n_RRC_SendProtocolPerChannel:=2;
    !
    TASK PERS num n_RRC_ReadPtrSenBufRob{n_RRC_NumOfCha}:=[8,1,1,1];
    TASK PERS num n_RRC_ReadPtrSenBufCtrl{n_RRC_NumOfCha}:=[1,1,1,1];
    !
    TASK PERS num n_RRC_SenHeaderSqzNr{n_RRC_NumOfCha}:=[17,0,0,0];
    !
    TASK PERS num n_RRC_SenMsgLenRob:=111;
    !
    TASK PERS num n_RRC_TimeStamp:=59.64;
    TASK PERS num n_RRC_TimeStampSec:=59;
    TASK PERS num n_RRC_TimeStampNanoSec:=639;

    !************************************************
    ! Declaration :     string
    !************************************************
    !
    TASK PERS string st_RRC_EvLogMsgHeader:="RRC -- Sender";
    !
    VAR string st_RRC_IP_ClientSen{n_RRC_NumOfCha}:=["","","",""];

    !************************************************
    ! Declaration :     clock
    !************************************************
    !
    VAR clock clk_RRC_TimeStamp;
    VAR clock clk_RRC_PackAndSend;

    !************************************************
    ! Declaration :     socketdev
    !************************************************
    !
    TASK VAR socketdev sod_RRC_ServerSen{n_RRC_NumOfCha};
    TASK VAR socketdev sod_RRC_ClientSen{n_RRC_NumOfCha};

    !************************************************
    ! Declaration :     RRC_Protokol
    !************************************************
    !
    CONST RRC_Protocol proEmpty:=[[0,0,0,0],[0,0,0,"",0,0,"",0,0,0,"",0,"",0,"",0,"",0,"",0,"",0,"",0,"",0,0,0,0,0,0,0,0,0,0,0,0,0,0,0,0,0,0,0,0,0,0,0,0,0,0,0,0,0,0,0,0,0,0,0,0,0]];
    !
    !* TASK VAR RRC_Protocol pro_RRC_ActMsgRob:=[[0,0,0,0],[0,0,0,"",0,0,"",0,0,0,"",0,"",0,"",0,"",0,"",0,0,0,0,0,0,0,0,0,0,0,0,0,0,0,0,0,0,0,0,0,0,0,0,0,0,0,0,0,0,0]];
    !
    TASK PERS RRC_Protocol pro_RRC_ActMsgSen{n_RRC_SendProtocolPerChannel,n_RRC_NumOfCha}:=[
    [[[0,0,0,0],[0,0,0,"",0,0,"",0,0,0,"",0,"",0,"",0,"",0,"",0,"",0,"",0,"",0,0,0,0,0,0,0,0,0,0,0,0,0,0,0,0,0,0,0,0,0,0,0,0,0,0,0,0,0,0,0,0,0,0,0,0,0]],
    [[0,0,0,0],[0,0,0,"",0,0,"",0,0,0,"",0,"",0,"",0,"",0,"",0,"",0,"",0,"",0,0,0,0,0,0,0,0,0,0,0,0,0,0,0,0,0,0,0,0,0,0,0,0,0,0,0,0,0,0,0,0,0,0,0,0,0]],
    [[0,0,0,0],[0,0,0,"",0,0,"",0,0,0,"",0,"",0,"",0,"",0,"",0,"",0,"",0,"",0,0,0,0,0,0,0,0,0,0,0,0,0,0,0,0,0,0,0,0,0,0,0,0,0,0,0,0,0,0,0,0,0,0,0,0,0]],
    [[0,0,0,0],[0,0,0,"",0,0,"",0,0,0,"",0,"",0,"",0,"",0,"",0,"",0,"",0,"",0,0,0,0,0,0,0,0,0,0,0,0,0,0,0,0,0,0,0,0,0,0,0,0,0,0,0,0,0,0,0,0,0,0,0,0,0]]],

    [[[115,2,59,639],[17,0,15,"r_RRC_GetJoints",0,4,"Done",1,0,0,"",0,"",0,"",0,"",0,"",0,"",0,"",0,"",12,-24.4963,-17.8131,33.2614,-59.6898,-28.7042,56.3166,9E+9,9E+9,9E+9,9E+9,9E+9,9E+9,0,0,0,0,0,0,0,0,0,0,0,0,0,0,0,0,0,0,0,0,0,0,0,0]],
    [[0,0,0,0],[0,0,0,"",0,0,"",0,0,0,"",0,"",0,"",0,"",0,"",0,"",0,"",0,"",0,0,0,0,0,0,0,0,0,0,0,0,0,0,0,0,0,0,0,0,0,0,0,0,0,0,0,0,0,0,0,0,0,0,0,0,0]],
    [[0,0,0,0],[0,0,0,"",0,0,"",0,0,0,"",0,"",0,"",0,"",0,"",0,"",0,"",0,"",0,0,0,0,0,0,0,0,0,0,0,0,0,0,0,0,0,0,0,0,0,0,0,0,0,0,0,0,0,0,0,0,0,0,0,0,0]],
    [[0,0,0,0],[0,0,0,"",0,0,"",0,0,0,"",0,"",0,"",0,"",0,"",0,"",0,"",0,"",0,0,0,0,0,0,0,0,0,0,0,0,0,0,0,0,0,0,0,0,0,0,0,0,0,0,0,0,0,0,0,0,0,0,0,0,0]]]];

    !************************************************
    ! Declaration :     rawbytes
    !************************************************
    !
    TASK VAR rawbytes rb_RRC_SenTempBuffer;
    TASK VAR rawbytes rb_RRC_SenBufferMsgLen;
    TASK VAR rawbytes rb_RRC_SenBuffer;

    !************************************************
    ! Declaration :     RRC_buffer_msg
    !************************************************
    !
    CONST RRC_buffer_msg bmEmpty:=[[0,0,0,"",0,0,"",0,0,0,"",0,"",0,"",0,"",0,"",0,"",0,"",0,"",0,0,0,0,0,0,0,0,0,0,0,0,0,0,0,0,0,0,0,0,0,0,0,0,0,0,0,0,0,0,0,0,0,0,0,0,0],FALSE];

ENDMODULE

--- Backups/vIRB4600-40-2.55-RW11/RAPID/TASK4/SYSMOD/RRC_UserInteraction.sys ---
MODULE RRC_UserInteraction (SYSMODULE, NOSTEPIN)
    !***********************************************************************************
    !
    ! ETH Zurich / Robotic Fabrication Lab
    ! HIB C 13 / Stefano-Franscini-Platz 1
    ! CH-8093 Zurich
    !
    !***********************************************************************************
    !
    ! PROJECT     :  RRC - Rapid Robot Communication
    !
    ! FUNCTION    :  General Utilities Library
    !
    ! AUTHOR      :  Philippe Fleischmann
    !
    ! EMAIL       :  rrc@arch.ethz.ch
    !
    ! HISTORY     :  2019.02.22
    !
    ! Copyright   :  ETH Zurich (CH) 2019
    !                - Philippe Fleischmann
    !                - Michael Lyrenmann
    !                - Gonzalo Casas
    !
    ! License     :  This code base is governed by an EULA (End-User License Agreement)
    !                which you have received together with the software.
    !                You are not allowed to use the software on a real robots
    !                without a signed EULA.
    !
    !                A copy of the EULA content is in the controller task (T_CTRL).
    !
    !***********************************************************************************

    !************************************************
    ! Function    :     Teach Pendant (old FelxPendant) Message
    ! Programmer  :     Philippe Fleischmann
    ! Date        :     2019.02.22
    !***************** ETH Zurich *******************
    !
    PROC r_RRC_TPMsg(string stMsg)
        !
        ! Clear Msg Panel
        TPErase;
        !
        ! Msg for user
        TPWrite stMsg;
        !
        ! Time to read the Msg
        WaitTime n_RRC_TimeTPMsg;
        RETURN ;
    ERROR
        ! Placeholder for Error Code...
    ENDPROC

    !************************************************
    ! Function    :     Teach Pendant (old FelxPendant) Error Message
    ! Programmer  :     Philippe Fleischmann
    ! Date        :     2019.02.22
    !***************** ETH Zurich *******************
    !
    PROC r_RRC_TPErrMsg(num nErrno\switch StopTask\switch StopAllTasks)
        !
        ! Clear Msg Panel
        TPErase;
        !
        ! Write error number
        TPWrite "ERRNO = "\Num:=nErrno;
        !
        ! Stop task
        IF Present(StopTask) Stop;
        !
        ! Stop all normal tasks
        IF Present(StopAllTasks) Stop\AllMoveTasks;
        RETURN ;
    ERROR
        ! Placeholder for Error Code...
    ENDPROC

    !************************************************
    ! Function    :     Event Log Message
    ! Programmer  :     Philippe Fleischmann
    ! Date        :     2019.02.22
    !***************** ETH Zurich *******************
    !
    PROC r_RRC_EvLogMsg(string stHeader,string stMsg)
        !
        ! Msg for user
        ErrWrite\I,stHeader+" "+stMsg,"rLogMsg";
        RETURN ;
    ERROR
        ! Placeholder for Error Code...
    ENDPROC

    !************************************************
    ! Function    :     User interface message
    ! Programmer  :     Philippe Fleischmann
    ! Date        :     2019.02.22
    !***************** ETH Zurich *******************
    !
    FUNC string f_RRC_UIMsg(string stMsgHeader,string stMsgL1,\string stMsgL2,\string stMsgL3,\string stMsgL4,\string stMsgL5,string stBtn1\string stBtn2\string stBtn3\string stBtn4\string stBtn5,icondata icIcon)
        VAR num nAnswer;
        VAR string stMsg{5};
        VAR string stBtn{5};
        VAR string stAnswer;
        !
        ! Initialize variables
        stMsg:=["","","","",""];
        stBtn:=["","","","",""];
        !
        ! Load meassge
        stMsg{1}:=stMsgL1;
        IF Present(stMsgL2) stMsg{2}:=stMsgL2;
        IF Present(stMsgL3) stMsg{3}:=stMsgL3;
        IF Present(stMsgL4) stMsg{4}:=stMsgL4;
        IF Present(stMsgL5) stMsg{5}:=stMsgL5;
        !
        ! Load buttons
        stBtn{1}:=stBtn1;
        IF Present(stBtn2) stBtn{2}:=stBtn2;
        IF Present(stBtn3) stBtn{3}:=stBtn3;
        IF Present(stBtn4) stBtn{4}:=stBtn4;
        IF Present(stBtn5) stBtn{5}:=stBtn5;
        !
        ! Msg for user
        nAnswer:=UIMessageBox(
            \Header:=stMsgHeader
            \MsgArray:=stMsg
            \BtnArray:=stBtn
            \Icon:=icIcon);
        !
        ! handle user answer
        IF nAnswer=1 stAnswer:=stBtn{1};
        IF nAnswer=2 stAnswer:=stBtn{2};
        IF nAnswer=3 stAnswer:=stBtn{3};
        IF nAnswer=4 stAnswer:=stBtn{4};
        IF nAnswer=5 stAnswer:=stBtn{5};
        !
        ! Return user answer as string
        RETURN stAnswer;
    ERROR
        ! Placeholder for Error Code...
    ENDFUNC

    !************************************************
    ! Function    :     User interface numerical entry
    ! Programmer  :     Philippe Fleischmann
    ! Date        :     2019.02.22
    !***************** ETH Zurich *******************
    !
    FUNC num f_RRC_UINumEntry(string stMsgHeader,string stMsgL1,\string stMsgL2,\string stMsgL3,\string stMsgL4,\string stMsgL5,num nMin,num nMax,\num nDefault,icondata icIcon)
        VAR string stMsg{5};
        VAR num nAnswer;
        VAR num nInitValue;
        !
        ! Initialize variables
        stMsg:=["","","","",""];
        nInitValue:=nMin;
        !
        ! Load meassge
        stMsg{1}:=stMsgL1;
        IF Present(stMsgL2) stMsg{2}:=stMsgL2;
        IF Present(stMsgL3) stMsg{3}:=stMsgL3;
        IF Present(stMsgL4) stMsg{4}:=stMsgL4;
        IF Present(stMsgL5) stMsg{5}:=stMsgL5;
        !
        ! Use default value when present
        IF Present(nDefault) nInitValue:=nDefault;
        !
        ! Msg for user
        nAnswer:=Round(UINumEntry(
            \Header:=stMsgHeader
            \MsgArray:=stMsg
            \Icon:=icIcon
            \InitValue:=nInitValue
            \MinValue:=nMin
            \MaxValue:=nMax)\Dec:=1);
        !
        ! Return user answer as string
        RETURN nAnswer;
    ERROR
        ! Placeholder for Error Code...
    ENDFUNC


ENDMODULE

--- Backups/vIRB4600-40-2.55-RW11/SYSPAR/EIO.cfg ---
EIO:CFG_1.0:6:1::
#
INDUSTRIAL_NETWORK:

      -Name "PROFINET" -Connection "PROFINET Network"\
      -Label "PROFINET Controller/Device Network" -StationName ""
#
PROFINET_DRIVER:

      -Name "PROFINET_COMMON_DATA"
#
PROFINET_INTERNAL_DEVICE:

      -Name "PN_Internal_Device" -VendorName "ABB Robotics"\
      -ProductName "PROFINET Internal Device"
#
EIO_SIGNAL:

      -Name "di_1" -SignalType "DI" -Access "All"

      -Name "do_1" -SignalType "DO" -Access "All"

      -Name "gi_1" -SignalType "GI" -Access "All"

      -Name "go_1" -SignalType "GO" -Access "All"

      -Name "ai_1" -SignalType "AI" -Access "All" -MaxLog 10 -MinLog -10

      -Name "ao_1" -SignalType "AO" -Access "All" -MaxLog 10 -MinLog -10

      -Name "do_X" -SignalType "DO" -Access "All"

      -Name "do_Y" -SignalType "DO" -Access "All"

      -Name "do_Z" -SignalType "DO" -Access "All"
